Staubli VAL3: oldmaduofrme.pgx

program oldmaduofrme()
begin
  f1.trsf=lib:fr1.trsf
  t1.trsf=lib:t1.trsf
end
